DATA_BLOCK "DB_MaterialHandlingCell"
{ S7_Optimized_Access := 'TRUE' }
VERSION : 0.1
NON_RETAIN
"FB_MaterialHandlingCell"
BEGIN
END_DATA_BLOCK
